(* PLC project ammonium-nitrates, Generated TextualNotationConverter 1.0 *)
(* stored: creationDateTime 2025-07-30T12:00:00, modificationDateTime 2025-07-30T12:00:00 *)

FUNCTION_BLOCK ANALOG_IN
  VAR_INPUT
    Name : STRING;
    Description : STRING;
    Raw_Signal : REAL;
    PV_High : REAL;
    PV_Low : REAL;
    Scaling_Slope : REAL;
    Scaling_Offset : REAL;
    Alarm_Enable : BOOL;
  END_VAR
  VAR_OUTPUT
    PV : REAL;
    High_Alarm : BOOL;
    Low_Alarm : BOOL;
    General_Fault : BOOL;
  END_VAR

            
          
END_FUNCTION_BLOCK

FUNCTION_BLOCK BOOL_IN
  VAR_INPUT
    Name : STRING;
    Description : STRING;
    Bool_In : BOOL;
    Alarm_OnTrue : BOOL;
    Alarm_OnFalse : BOOL;
    Latch_Enable : BOOL;
    Reset_Latch : BOOL;
  END_VAR
  VAR_OUTPUT
    Bool_Out : BOOL;
    Alarm_Active : BOOL;
    Latched_Status : BOOL;
  END_VAR

            
          
END_FUNCTION_BLOCK

FUNCTION_BLOCK PID_BASIC
  VAR_INPUT
    Name : STRING;
    Description : STRING;
    AUTO : BOOL;
    PV : REAL;
    SP : REAL;
    MV_MIN : REAL;
    MV_MAX : REAL;
    X0 : REAL;
    KP : REAL;
    TR : REAL;
    TD : REAL;
    PV_High : REAL;
    PV_Low : REAL;
    Deviation_Limit : REAL;
    Inhibit : BOOL;
  END_VAR
  VAR_OUTPUT
    PV_High_Alarm : BOOL;
    PV_Low_Alarm : BOOL;
    Deviation_Alarm : BOOL;
    XOUT : REAL;
  END_VAR

            
          
END_FUNCTION_BLOCK

FUNCTION_BLOCK RATIO_CONTROL
  VAR_INPUT
    Name : STRING;
    Description : STRING;
    Auto : BOOL;
    PrimaryPV : REAL;
    SecondaryPV : REAL;
    RatioSP : REAL;
    Bias : REAL;
    TrimKp : REAL;
    TrimTi : STRING;
    MV_MIN : REAL;
    MV_MAX : REAL;
    ManOut : REAL;
    Inhibit : BOOL;
  END_VAR
  VAR_OUTPUT
    SlaveSP : REAL;
    ActiveRatio : REAL;
    RatioErr : REAL;
  END_VAR

            
          
END_FUNCTION_BLOCK

FUNCTION_BLOCK VALVE_ELECTRIC
  VAR_INPUT
    Name : STRING;
    Description : STRING;
    Control_Signal : REAL;
    Manual_Mode : BOOL;
    Manual_Position : REAL;
    Open_Limit : REAL;
    Close_Limit : REAL;
    Timeout : STRING;
    Inhibit : BOOL;
  END_VAR
  VAR_OUTPUT
    Valve_Position : REAL;
    Feedback_Pos : REAL;
    Valve_Moving : BOOL;
    Position_Error : BOOL;
    Alarm : BOOL;
  END_VAR

            
          
END_FUNCTION_BLOCK

PROGRAM Section2
  VAR
    FT101_AmmoniaFlow_PV : REAL;
    FT102_AcidFlow_PV : REAL;
    LT104_Level_PV : REAL;
    PH105_pH_PV : REAL;
    FFIC102_AcidFlow_SP : REAL;
    FFIC102_Active_Ratio : REAL;
    VS107_Running : BOOL;
  END_VAR
  VAR
    FT-101 : ANALOG_IN;
    FT-102 : ANALOG_IN;
    LT-104 : ANALOG_IN;
    PH-105 : ANALOG_IN;
    FIC-101 : PID_BASIC;
    FIC-102 : PID_BASIC;
    TIC-103 : PID_BASIC;
    FV-101 : VALVE_ELECTRIC;
    FV-102 : VALVE_ELECTRIC;
    FFIC-102 : RATIO_CONTROL;
    VS-107 : BOOL_IN;
  END_VAR
  VAR  (* added by the conversion: wires and edge detectors of the diagram *)
    _OR1_OUT : BOOL;
  END_VAR

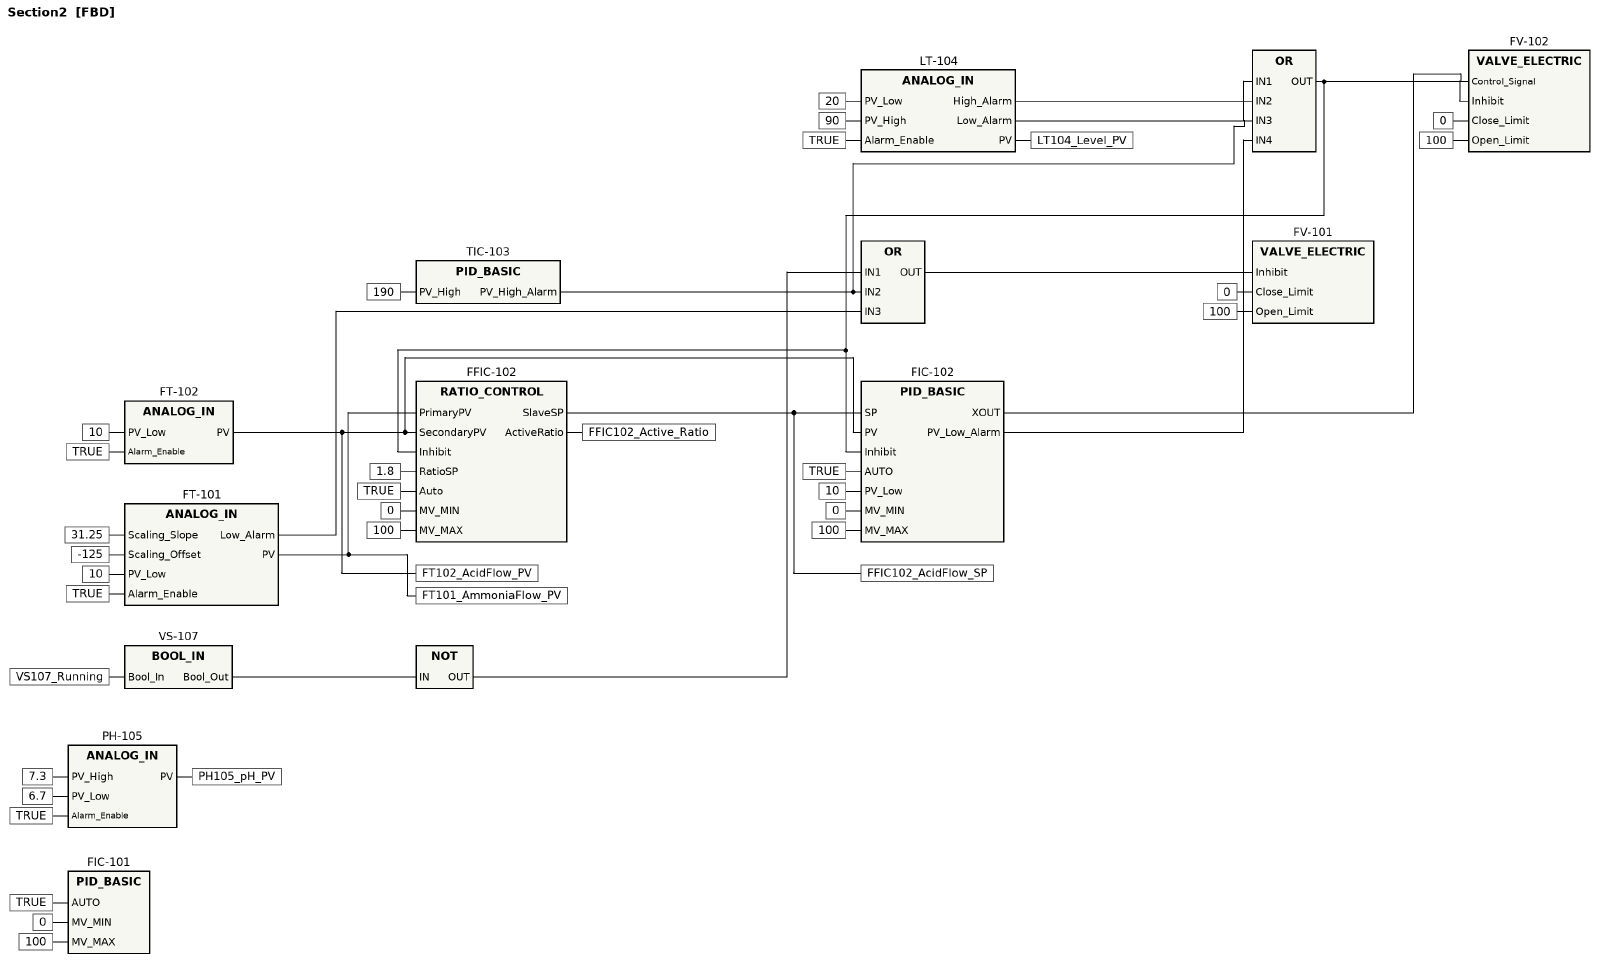
(* FBD diagram, written out as Structured Text *)
FT-101(Scaling_Slope := 31.25, Scaling_Offset := -125, PV_Low := 10, Alarm_Enable := TRUE);
FT-102(PV_Low := 10, Alarm_Enable := TRUE);
LT-104(PV_Low := 20, PV_High := 90, Alarm_Enable := TRUE);
TIC-103(PV_High := 190);
FIC-102(SP := FFIC-102.SlaveSP, PV := FT-102.PV, Inhibit := _OR1_OUT, AUTO := TRUE, PV_Low := 10, MV_MIN := 0, MV_MAX := 100);
_OR1_OUT := LT-104.Low_Alarm OR LT-104.High_Alarm OR TIC-103.PV_High_Alarm OR FIC-102.PV_Low_Alarm;
FFIC-102(PrimaryPV := FT-101.PV, SecondaryPV := FT-102.PV, Inhibit := _OR1_OUT, RatioSP := 1.8, Auto := TRUE, MV_MIN := 0, MV_MAX := 100);
FFIC102_AcidFlow_SP := FFIC-102.SlaveSP;
FFIC102_Active_Ratio := FFIC-102.ActiveRatio;
FT101_AmmoniaFlow_PV := FT-101.PV;
FT102_AcidFlow_PV := FT-102.PV;
LT104_Level_PV := LT-104.PV;
PH-105(PV_High := 7.3, PV_Low := 6.7, Alarm_Enable := TRUE);
PH105_pH_PV := PH-105.PV;
VS-107(Bool_In := VS107_Running);
FIC-101(AUTO := TRUE, MV_MIN := 0, MV_MAX := 100);
FV-101(Inhibit := NOT VS-107.Bool_Out OR TIC-103.PV_High_Alarm OR FT-101.Low_Alarm, Close_Limit := 0, Open_Limit := 100);
FV-102(Control_Signal := FIC-102.XOUT, Inhibit := _OR1_OUT, Close_Limit := 0, Open_Limit := 100);
END_PROGRAM

FUNCTION_BLOCK DIGITAL_IN
  VAR_INPUT
    Name : STRING;
    Description : STRING;
    DI_Raw : BOOL;
    DebounceTime : STRING;
    EnableAlarm : BOOL;
  END_VAR
  VAR_OUTPUT
    DI_Out : BOOL;
    Fault_State : BOOL;
  END_VAR

            
          
END_FUNCTION_BLOCK

FUNCTION_BLOCK DUTY_STANDBY
  VAR_INPUT
    Name : STRING;
    Description : STRING;
    Enable : BOOL;
    StartRequest : BOOL;
    AlternateEnable : BOOL;
    ForcePumpA : BOOL;
    ForcePumpB : BOOL;
    DutyElapsed : BOOL;
    MinRunElapsed : BOOL;
    SwitchoverDelayElapsed : BOOL;
    StartTimeoutElapsed : BOOL;
    PumpA_RunFB : BOOL;
    PumpB_RunFB : BOOL;
    PumpA_Fault : BOOL;
    PumpB_Fault : BOOL;
    Reset : BOOL;
    Inhibit : BOOL;
  END_VAR
  VAR_OUTPUT
    CmdPumpA : BOOL;
    CmdPumpB : BOOL;
    ActiveIsA : BOOL;
    SwitchedDueToDuty : BOOL;
    SwitchedDueToFailure : BOOL;
    Alarm_FailedStart_A : BOOL;
    Alarm_FailedStart_B : BOOL;
    Alarm_NoAvailablePump : BOOL;
  END_VAR

            
          
END_FUNCTION_BLOCK

FUNCTION_BLOCK MOTOR_2SPD
  VAR_INPUT
    Name : STRING;
    Description : STRING;
    Start_Cmd : BOOL;
    Stop_Cmd : BOOL;
    Speed_High_Cmd : BOOL;
    Speed_Low_Cmd : BOOL;
    Inhibit : BOOL;
  END_VAR
  VAR_OUTPUT
    Motor_Start_Out : BOOL;
    FB_Running : BOOL;
    FB_Trip : BOOL;
    FB_HighSpeed : BOOL;
    FB_LowSpeed : BOOL;
    Alarm_Speed_Error : BOOL;
  END_VAR

            
          
END_FUNCTION_BLOCK

FUNCTION_BLOCK MOTOR_ON_OFF
  VAR_INPUT
    Name : STRING;
    Description : STRING;
    Start_Cmd : BOOL;
    Stop_Cmd : BOOL;
    Start_Delay : STRING;
    MinRunTime : STRING;
    Inhibit : BOOL;
  END_VAR
  VAR_OUTPUT
    Motor_Start_Out : BOOL;
    FB_Running : BOOL;
    FB_Trip : BOOL;
    Alarm_Start_Fail : BOOL;
    Alarm_Stop_Fail : BOOL;
  END_VAR

            
          
END_FUNCTION_BLOCK

FUNCTION_BLOCK MOTOR_VSD
  VAR_INPUT
    Name : STRING;
    Description : STRING;
    Start_Cmd : BOOL;
    Stop_Cmd : BOOL;
    Speed_SP : REAL;
    Accel_Ramp : STRING;
    Decel_Ramp : STRING;
    Inhibit : BOOL;
  END_VAR
  VAR_OUTPUT
    Speed_Out : REAL;
    FB_Running : BOOL;
    FB_Fault : BOOL;
    FB_Ready : BOOL;
    FB_ActualSpeed : REAL;
    Alarm_Speed_Deviation : BOOL;
    Alarm_Comm_Fail : BOOL;
  END_VAR

            
          
END_FUNCTION_BLOCK

FUNCTION_BLOCK SPLIT_RANGE
  VAR_INPUT
    Name : STRING;
    Description : STRING;
    IN : REAL;
    Split_Point : REAL;
    Output1_Start : REAL;
    Output1_End : REAL;
    Output2_Start : REAL;
    Output2_End : REAL;
  END_VAR
  VAR_OUTPUT
    OUT1 : REAL;
    OUT2 : REAL;
  END_VAR

            
          
END_FUNCTION_BLOCK

FUNCTION_BLOCK VALVE_ON_OFF
  VAR_INPUT
    Name : STRING;
    Description : STRING;
    Open_Cmd : BOOL;
    Close_Cmd : BOOL;
    Timeout : STRING;
    Inhibit : BOOL;
  END_VAR
  VAR_OUTPUT
    FB_Opened : BOOL;
    FB_Closed : BOOL;
    Valve_Open_Out : BOOL;
    Valve_Close_Out : BOOL;
    Alarm_Position_Error : BOOL;
    Alarm_General : BOOL;
  END_VAR

            
          
END_FUNCTION_BLOCK

FUNCTION_BLOCK VOTING_ANALOG
  VAR_INPUT
    Name : STRING;
    Description : STRING;
    Input1 : REAL;
    Input2 : REAL;
    Input3 : REAL;
    Deviation_Limit : REAL;
    Voting_Scheme : STRING;
    EnableAlarm : BOOL;
    Inhibit : BOOL;
  END_VAR
  VAR_OUTPUT
    Voted_Output : REAL;
    Sensor1_Fault : BOOL;
    Sensor2_Fault : BOOL;
    Sensor3_Fault : BOOL;
    Alarm_Voting_Error : BOOL;
    Healthy_Sensors_Count : INT;
  END_VAR

            
          
END_FUNCTION_BLOCK

CONFIGURATION Config0
  RESOURCE Res0 ON PLC
    TASK task0(INTERVAL := T#20ms, PRIORITY := 0);
    PROGRAM instance0 WITH task0 : Section2;
  END_RESOURCE
END_CONFIGURATION
